FUNCTION_BLOCK PUBLIC EventEmitter_TestSuit EXTENDS TcUnit.FB_TestSuite
VAR
END_VAR

CheckEmitWorksWithHandler();
CheckEmitWorksWithMultipleHandlers();
CheckEventIsNotSentToTheWrongHandler();
CheckOffEventUnregistersAHandler();
CheckClearUnregistersMultipleHandlers();

METHOD PUBLIC CheckClearUnregistersMultipleHandlers
VAR
	mockEvent : MockEvent;
	mockHandler1 : MockEventHandler;
	mockHandler2 : MockEventHandler;
	eventEmitter : EventEmitter;
	eventReceived : BOOL;
END_VAR
TEST('CheckClearUnregistersMultipleHandlers');

// @TEST-FIXTURE
eventEmitter.OnEvent('test', mockHandler1);
eventEmitter.OnEvent('test', mockHandler2);
eventEmitter.Clear();

// @TEST-RUN
eventEmitter.Emit('test',mockEvent);
eventReceived := mockHandler1.EqualsLastEvent(mockEvent) OR mockHandler2.EqualsLastEvent(mockEvent) ;

// @TEST-ASSSERT
AssertFalse(
	Condition := eventReceived,
	Message := 'Event Emitter did not correctly unregister multiple handlers following a clear'
);

TEST_FINISHED();
END_METHOD

METHOD PUBLIC CheckEmitWorksWithHandler
VAR
	mockEvent : MockEvent;
	mockHandler : MockEventHandler;
	eventEmitter : EventEmitter;
	eventReceived : BOOL;
END_VAR
TEST('CheckEmitWorksWithHandler');

// @TEST-FIXTURE
eventEmitter.OnEvent('test', mockHandler);

// @TEST-RUN
eventEmitter.Emit('test',mockEvent);
eventReceived := mockHandler.EqualsLastEvent(mockEvent);

// @TEST-ASSSERT
AssertTrue(
	Condition := eventReceived,
	Message := 'Event Emitter did not correctly emmit the event to the handler'
);

TEST_FINISHED();
END_METHOD

METHOD PUBLIC CheckEmitWorksWithMultipleHandlers
VAR
	mockEvent : MockEvent;
	mockHandler1 : MockEventHandler;
	mockHandler2 : MockEventHandler;
	eventEmitter : EventEmitter;
	eventReceived : BOOL;
END_VAR
TEST('CheckEmitWorksWithMultipleHandlers');

// @TEST-FIXTURE
eventEmitter.OnEvent('test', mockHandler1);
eventEmitter.OnEvent('test', mockHandler2);

// @TEST-RUN
eventEmitter.Emit('test',mockEvent);
eventReceived := mockHandler1.EqualsLastEvent(mockEvent) AND mockHandler2.EqualsLastEvent(mockEvent) ;

// @TEST-ASSSERT
AssertTrue(
	Condition := eventReceived,
	Message := 'Event Emitter did not correctly emmit the event to multiple handlers'
);

TEST_FINISHED();
END_METHOD

METHOD PUBLIC CheckEventIsNotSentToTheWrongHandler
VAR
	mockEvent : MockEvent;
	mockHandler : MockEventHandler;
	eventEmitter : EventEmitter;
	eventReceived : BOOL;
END_VAR
TEST('CheckEventIsNotSentToTheWrongHandler');

// @TEST-FIXTURE
eventEmitter.OnEvent('foo', mockHandler);

// @TEST-RUN
eventEmitter.Emit('bar',mockEvent);
eventReceived := mockHandler.EqualsLastEvent(mockEvent);

// @TEST-ASSSERT
AssertFalse(
	Condition := eventReceived,
	Message := 'Event Emitter sent the event to the wrong handler'
);

TEST_FINISHED();
END_METHOD

METHOD PUBLIC CheckOffEventUnregistersAHandler
VAR
	mockEvent : MockEvent;
	mockHandler : MockEventHandler;
	eventEmitter : EventEmitter;
	eventReceived : BOOL;
END_VAR
TEST('CheckOffEventUnregistersAHandler');

// @TEST-FIXTURE
eventEmitter.OnEvent('test', mockHandler);
eventEmitter.OffEvent('test', mockHandler);

// @TEST-RUN
eventEmitter.Emit('test',mockEvent);
eventReceived := mockHandler.EqualsLastEvent(mockEvent);

// @TEST-ASSSERT
AssertFalse(
	Condition := eventReceived,
	Message := 'Event Emitter did not correctly unregister the event handler using the off method'
);

TEST_FINISHED();
END_METHOD

END_FUNCTION_BLOCK

(* stored: Version 1.1.0.1, ProductVersion 3.1.4024.12
   POU EventEmitter_TestSuit: Id {c771dd79-b70b-0181-1b27-c5e2c81ee9a4}, SpecialFunc None
   Method CheckClearUnregistersMultipleHandlers: Id {6f968a81-0a57-03c6-3348-3b3f43b11e67}
   Method CheckEmitWorksWithHandler: Id {2e5817dc-28f3-0522-2aca-21ad8e95462f}
   Method CheckEmitWorksWithMultipleHandlers: Id {ca286491-29ce-0ee7-232d-791d78869866}
   Method CheckEventIsNotSentToTheWrongHandler: Id {c9d6842b-c5e0-0fa4-11db-eb3e4bccea3b}
   Method CheckOffEventUnregistersAHandler: Id {0291f32e-8068-0b28-38a8-cb83a2bc5dca} *)
